FUNCTION_BLOCK StopMoverGroup EXTENDS TaskBase
VAR_INPUT
END_VAR
VAR_OUTPUT
END_VAR
VAR
	groupStop			: MC_GroupStop;
	_caGroup			: ICollisionGroup;
	_stopGroup : BOOL;
	_jerk : MC_LREAL;
	_deceleration : MC_LREAL;
	Logger : TcMessage_Ext;
END_VAR

{analysis -2}

METHOD Abort : BOOL
groupStop.Execute := FALSE;
State := 0;
Abort := true;
END_METHOD

METHOD Cycle : HRESULT
VAR_INPUT
END_VAR
Cycle := S_OK;
CASE State OF
	0:
		IF _stopGroup THEN
			Cycle := S_PENDING;
			_Done := FALSE;
			_Error := FALSE;
			_Busy := TRUE;
			groupStop.Execute := TRUE;
			IF groupStop.Busy THEN
				State := 10;
				_stopGroup := FALSE;
				Logger.Send(TC_EVENTS.XtsCaGroupEvents.CAGroupStopping,'');
			END_IF
		END_IF
	10:
		IF groupStop.Done THEN
			_Done := TRUE;
			Logger.Send(TC_EVENTS.XtsCaGroupEvents.CAGroupStopped,'');
		ELSIF groupStop.Error THEN
			_Error := TRUE;
			Logger.Send(TC_EVENTS.XtsCaGroupEvents.CAGroupStopError,'');
		END_IF
		IF _Done OR _Error THEN
			_Busy := FALSE;
			groupStop.Execute := FALSE;
			State := 0;
			Cycle := S_OK;
		END_IF
	ELSE
		Cycle := E_FAIL;
END_CASE


groupStop(AxesGroup := _caGroup.GroupRef);
END_METHOD

PROPERTY PUBLIC Deceleration : MC_LREAL
GET
Deceleration := _deceleration;
END_GET
SET
_deceleration := Deceleration;
END_SET
END_PROPERTY

METHOD Execute : BOOL
_stopGroup := Execute := true;
END_METHOD

METHOD FB_init : BOOL
VAR_INPUT
	bInitRetains : BOOL; // if TRUE, the retain variables are initialized (warm start / cold start)
	bInCopyCode : BOOL;  // if TRUE, the instance afterwards gets moved into the copy code (online change)
	CAGroup : ICollisionGroup;
END_VAR
_caGroup := CAGroup;
END_METHOD

PROPERTY PUBLIC Jerk : MC_LREAL
GET
Jerk := _jerk;
END_GET
SET
_jerk := Jerk;
END_SET
END_PROPERTY

END_FUNCTION_BLOCK

(* stored: Version 1.1.0.1, ProductVersion 3.1.4024.12
   POU StopMoverGroup: Id {1c1e07aa-be1f-4f5f-9f83-11f52cae0c47}, SpecialFunc None
   Method Abort: Id {c537197c-b147-4abf-b878-34be8d4864fb}
   Method Cycle: Id {eb283c73-ef4f-42f6-83b9-10b77e01e97b}
   Property Deceleration: Id {4b0f086c-1d53-44e4-86b9-9d4a701184a7}
   Get Get: Id {b0811cfb-bb5c-42b5-9a5c-793a076794d1}
   Set Set: Id {d5d2a280-9e98-49b7-b6fe-a592814414dd}
   Method Execute: Id {699db21e-cd5b-48cd-b391-3ef65bad1290}
   Method FB_init: Id {4499cf15-952b-423e-bc0b-2b67686c6e93}
   Property Jerk: Id {753822d2-3240-4ac1-a838-285435826cfe}
   Get Get: Id {8ec059f8-9a70-4be4-bfe0-899344b2368e}
   Set Set: Id {1e87f5ff-9029-43fd-96bd-fd5c4e284768} *)
